{attribute 'linkalways'} 
{attribute 'no_explicit_call' := 'This FB is a CLASS and must be accessed using methods or properties'}
{attribute 'enable_dynamic_creation'}
FUNCTION_BLOCK Node_F_VN_ContainerAverageVarianceElementwise2 EXTENDS VisionNode
VAR
    ipSrcContainer : _ITcVnContainer;
    aAverage : _TcVnVector2_LREAL;
	aVariance : _TcVnVector2_LREAL;
    hrPrev : _HRESULT(S_OK);
    hresult : _HRESULT(S_OK);
END_VAR

METHOD PUBLIC  Clone : I_Node
VAR
	pNode : POINTER TO Node_F_VN_ContainerAverageVarianceElementwise2;
END_VAR
pNode := __NEW(Node_F_VN_ContainerAverageVarianceElementwise2);
Clone := pNode^;
END_METHOD

METHOD FB_init : BOOL
VAR_INPUT
	bInitRetains : BOOL; // if TRUE, the retain variables are initialized (warm start / cold start)
	bInCopyCode : BOOL;  // if TRUE, the instance afterwards gets moved into the copy code (online change)
END_VAR
AddInput('ipSrcContainer', ipSrcContainer);
AddInput('hrPrev', hrPrev);
AddOutput('aAverage', aAverage);
AddOutput('aVariance', aVariance);
AddOutput('hresult',hresult);
END_METHOD

METHOD PROTECTED OnExecute
hresult.Value := F_VN_ContainerAverageVarianceElementwise2(
    ipSrcContainer := ipSrcContainer.Value,
    aAverage := aAverage.Value,
	aVariance := aVariance.Value,
    hrPrev:= hrPrev.Value);
END_METHOD

METHOD PUBLIC PreExecutionCheck
VAR_INPUT
	Check : I_PreExecutionChecks;
END_VAR
VAR
	isCorrectType : BOOL;
END_VAR
Check.IsTrue(ipSrcContainer.IsValid, 'ipContainer must be a valid container');

isCorrectType := 
    // ---------------------------------------------------------
    // Point 2 Types (X, Y)
    // ---------------------------------------------------------
    ipSrcContainer.IsType(TC_GLOBAL_CONST_LIST.ContainerType_Vector_TcVnPoint2_DINT) OR_ELSE
    ipSrcContainer.IsType(TC_GLOBAL_CONST_LIST.ContainerType_Vector_TcVnPoint2_REAL) OR_ELSE
    ipSrcContainer.IsType(TC_GLOBAL_CONST_LIST.ContainerType_Vector_TcVnPoint2_LREAL) OR_ELSE

    // ---------------------------------------------------------
    // Vector 2 Types (X, Y)
    // ---------------------------------------------------------
    ipSrcContainer.IsType(TC_GLOBAL_CONST_LIST.ContainerType_Vector_TcVnVector2_SINT) OR_ELSE
    ipSrcContainer.IsType(TC_GLOBAL_CONST_LIST.ContainerType_Vector_TcVnVector2_USINT) OR_ELSE
    ipSrcContainer.IsType(TC_GLOBAL_CONST_LIST.ContainerType_Vector_TcVnVector2_INT) OR_ELSE
    ipSrcContainer.IsType(TC_GLOBAL_CONST_LIST.ContainerType_Vector_TcVnVector2_UINT) OR_ELSE
    ipSrcContainer.IsType(TC_GLOBAL_CONST_LIST.ContainerType_Vector_TcVnVector2_DINT) OR_ELSE
    ipSrcContainer.IsType(TC_GLOBAL_CONST_LIST.ContainerType_Vector_TcVnVector2_REAL);

Check.IsTrue(isCorrectType, 'ipContainer contains incorrect type for Elementwise2');
END_METHOD

END_FUNCTION_BLOCK

(* stored: Version 1.1.0.1, ProductVersion 3.1.4026.13
   POU Node_F_VN_ContainerAverageVarianceElementwise2: Id {ebd80e81-7a63-08aa-1784-06486dc139e7}, SpecialFunc None
   Folder Constructor: Id {f119bff7-8c31-0310-2d55-342e3633d97d}
   Method Clone: Id {805679ec-914b-060f-0c3d-7adb93731beb}
   Method FB_init: Id {d51396e7-5336-0dc7-2cfe-74334b1ff748}
   Method OnExecute: Id {19eba451-a7ad-0226-025a-5c7d063608dc}
   Method PreExecutionCheck: Id {84e05b40-f1c2-0d28-215f-c9d3e2c78f35} *)
